(* Logix 5000 project; controller Comas_L4 vendor 1 type 14 code 193 rev 30.11; software revision 30.02; part 11 of 12 *)
(* tags used below, declared in another part *)
   AOI_Badge : Badges_Acces;
   AOI_Cam_Display_Horiz : AOI_CamDisplay_OCX_StdCAM;
   AOI_Cam_Display_Verti : AOI_CamDisplay_OCX_StdCAM;
   AOI_Pilotage_Codeur_Vitesse_Moy : Pilotage_Vitesse_Rapide_V4;
   Axe_Codeur_Four : AXIS_CIP_DRIVE;
   Axe_Horizontal_Gauche : AXIS_CIP_DRIVE;
   Axe_Virtuel_Codeur : AXIS_VIRTUAL;
   Axe_Virtuel_Maitre : AXIS_VIRTUAL;
   Badge_Code_A : BOOL;
   Badge_Code_B : BOOL;
   Badge_Code_C : BOOL;
   Badge_Code_D : BOOL;
   BP_O_F_Trappe : BOOL;
   Cam_Chart_Horiz : Chart;
   Cam_Chart_Verti : Chart;
   Cam_Display_Horiz : UDT_Axis_Cam_Profil;
   Cam_Display_Verti : UDT_Axis_Cam_Profil;
   CO_Acquit_defaut : BOOL;
   CO_Defaut_Four : BOOL;
   CO_Defaut_Relais_Securite : BOOL;
   CO_Defauts_Secondaires : BOOL;
   CO_demande_darret : BOOL;
   CO_en_Marche : BOOL;
   CO_Engage_Axe_H_Droit : Engage_Axe;
   CO_Engage_Axe_H_Gauche : Engage_Axe;
   CO_Engage_Axe_V_Droit : Engage_Axe;
   CO_Engage_Axe_V_Gauche : Engage_Axe;
   CO_Engage_Maitre : Engage_Axe_Virtuel;
   CO_Engagement : BOOL;
   CO_Flip_100ms : TIMER;
   CO_Flip_500ms : TIMER;
   CO_Flop_100ms : TIMER;
   CO_Flop_500ms : TIMER;
   CO_Init_Ok : BOOL;
   CO_Machine_sans_defaut : BOOL;
   CO_Marche : BOOL;
   CO_Pilotage_Coupe_Fil : Pilotage_Relatif_Virtuel;
   CO_Synchro_Axe_En_Cours : BOOL;
   CO_Temps_de_demarrage : TIMER;
   CO_TOF_Top_Decoreuse : TIMER;
   CO_TOF_Top_Doseuse : TIMER;
   CO_Top_Debut_Cycle_Decoreuse : BOOL;
   CO_Top_Debut_Dosage : BOOL;
   CO_Top_Once_Decoreuse : BOOL;
   CO_Top_Once_Doseuse : BOOL;
   CO_Top_Recalage : BOOL;
   Com_Comas_Conv : DINT[10];
   Com_Comas_Gen_Conv : DINT[10];
   Com_Comas_Sortie_F : UDT_COM_Comas_Vers_SortieF;
   Det_Produit : BOOL;
   Det_Produit2 : BOOL;
   ENT_Badge_Code_A : ALIAS FOR Local:1:I.Pt11.Data;
   ENT_Badge_Code_B : ALIAS FOR Local:1:I.Pt12.Data;
   ENT_Badge_Code_C : ALIAS FOR Local:1:I.Pt13.Data;
   ENT_Badge_Code_D : ALIAS FOR Local:1:I.Pt14.Data;
   ENT_Badge_STR : ALIAS FOR Local:1:I.Pt15.Data;
   ENT_CO_BP_Arret : ALIAS FOR Local:1:I.Pt01.Data;
   ENT_CO_BP_Marche : ALIAS FOR Local:1:I.Pt00.Data;
   ENT_Reisdorf_en_Marche : ALIAS FOR Local:2:I.Pt03.Data;
   Fin_Rouleau : REAL;
   Flip_Display : TIMER;
   Flop_Display : TIMER;
   Front_Badge : BOOL;
   Front_Det_produit_Moyennage : BOOL;
   Front_Det_produit_Moyennage2 : BOOL;
   Front_Resynchro_temp : BOOL;
   Front_Top_Recalage : BOOL;
   Lecteur_Badge_Code_A : BOOL;
   Lecteur_Badge_Code_B : BOOL;
   Lecteur_Badge_Code_C : BOOL;
   Lecteur_Badge_Code_D : BOOL;
   MAM_Resyncho_Codeur : MOTION_INSTRUCTION;
   MAM_Resynchro_Accel_Correction : REAL;
   MAM_Resynchro_Vitesse_Correction : REAL;
   Memo_Recalage_Detection_PRoduit_1 : BOOL;
   Memo_Recalage_Detection_PRoduit_2 : BOOL;
   MSG_General_Convoyage : MESSAGE;
   MSG_Vitesse_Four_L4 : MESSAGE;
   Output_Cams_Decoreuse : Output_Cams;
   Output_Cams_Dosage : Output_Cams;
   Output_Cams_Recalage : Output_Cams;
   PCAM_Horizontal : UDT_CamGeneration;
   PCAM_Vertical : UDT_CamGeneration;
   Position_Codeur_Virtuel_Det_Produit : REAL;
   Position_Decalee : REAL;
   RECETTE_EC : UDT_RECIPE;
   Resynchro_Codeur : BOOL;
   Resynchro_Codeur_Front : BOOL;
   RSW_BADGE_Numero_Page : DINT;
   RSW_BADGE_Numero_Page_En_Cours : DINT;
   RSW_BADGE_RAZ_CODE : BOOL;
   RSW_BADGE_Temps_Restant : DINT;
   RSW_BADGE_TOF_Chagement_Page : TIMER;
   RSW_Niveau_Accu_LA : DINT;
   RSW_Niveau_Accu_LD : DINT;
   SOR_CO_Echange_Amont_OK : ALIAS FOR Local:3:O.Pt07.Data;
   SOR_CO_Top_Debut_Cycle_Decoreuse : ALIAS FOR Local:3:O.Pt05.Data;
   SOR_CO_Top_Debut_Dosage : ALIAS FOR Local:3:O.Pt06.Data;
   SOR_CO_Voyant_Arret : ALIAS FOR Local:3:O.Pt01.Data;
   SOR_CO_Voyant_Marche : ALIAS FOR Local:3:O.Pt00.Data;
   SOR_CO_Voyant_Rearmement : ALIAS FOR Local:3:O.Pt02.Data;
   Speed_Control_Pompe : Axis_speed_control;
   Start_Cam_Logique_Rouleaux : REAL;
   Stop_Cam_Logique_Rouleaux : REAL;
   Tab_Position_Correction : REAL[50];
   Tab_Position_Correction_Temp : REAL[50];
   Temps_total_avant_arret_L4 : REAL;
   TimeOutResynch_Codeur : TIMER;
   TON_Simul_Produit : TIMER;
   Val_Position_Recalage : REAL;
   Val_Position_Recalage_Tab1 : REAL;
   Val_Position_Recalage_Tab2 : REAL;
   Val_Position_Recalage_Tab3 : REAL;
   Val_Position_Recalage_Tab4 : REAL;
   Val_Position_Recalage_Tab5 : REAL;
   Vitesse_Four4_Real : REAL;
(* General, continued *)

ROUTINE D00_Marche   (* ladder *)
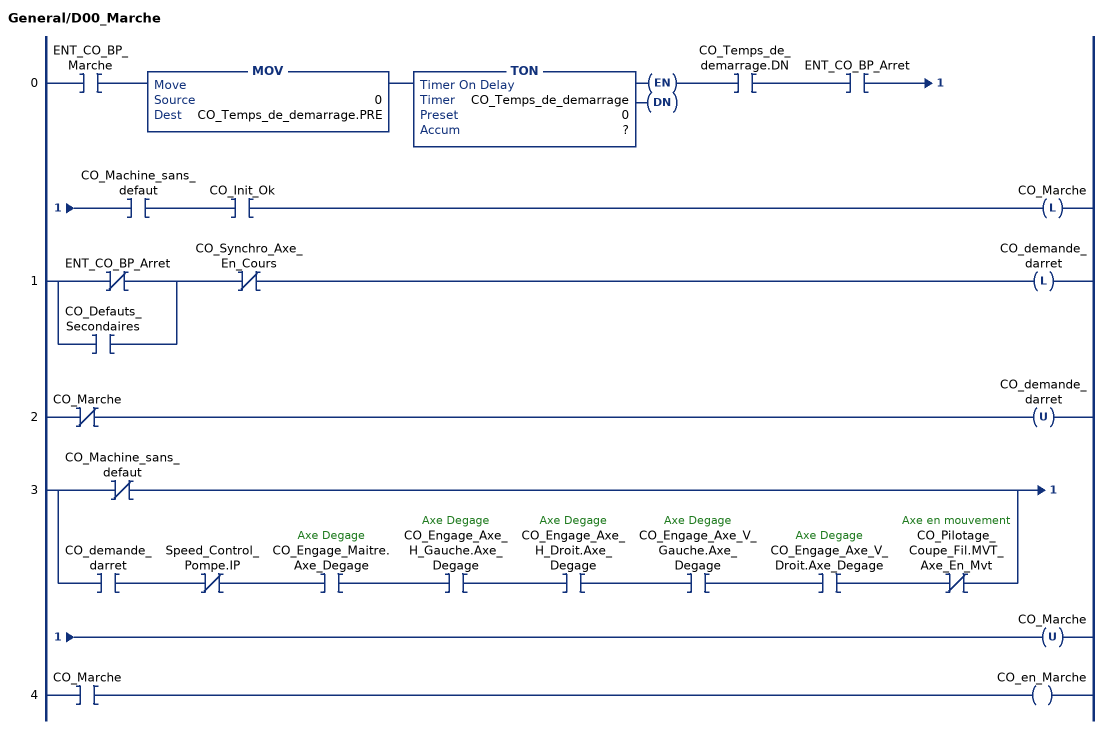
   0: XIC(ENT_CO_BP_Marche)MOV(0,CO_Temps_de_demarrage.PRE)TON(CO_Temps_de_demarrage,?,?)XIC(CO_Temps_de_demarrage.DN)XIC(ENT_CO_BP_Arret)XIC(CO_Machine_sans_defaut)XIC(CO_Init_Ok)OTL(CO_Marche);
   1: [XIO(ENT_CO_BP_Arret) ,XIC(CO_Defauts_Secondaires) ]XIO(CO_Synchro_Axe_En_Cours)OTL(CO_demande_darret);
   2: XIO(CO_Marche)OTU(CO_demande_darret);
   3: [XIO(CO_Machine_sans_defaut) ,XIC(CO_demande_darret) XIO(Speed_Control_Pompe.IP) XIC(CO_Engage_Maitre.Axe_Degage) XIC(CO_Engage_Axe_H_Gauche.Axe_Degage) XIC(CO_Engage_Axe_H_Droit.Axe_Degage) XIC(CO_Engage_Axe_V_Gauche.Axe_Degage) XIC(CO_Engage_Axe_V_Droit.Axe_Degage) XIO(CO_Pilotage_Coupe_Fil.MVT_Axe_En_Mvt) ]OTU(CO_Marche);
   4: XIC(CO_Marche)OTE(CO_en_Marche);
END_ROUTINE

ROUTINE E00_Voyants   (* ladder *)
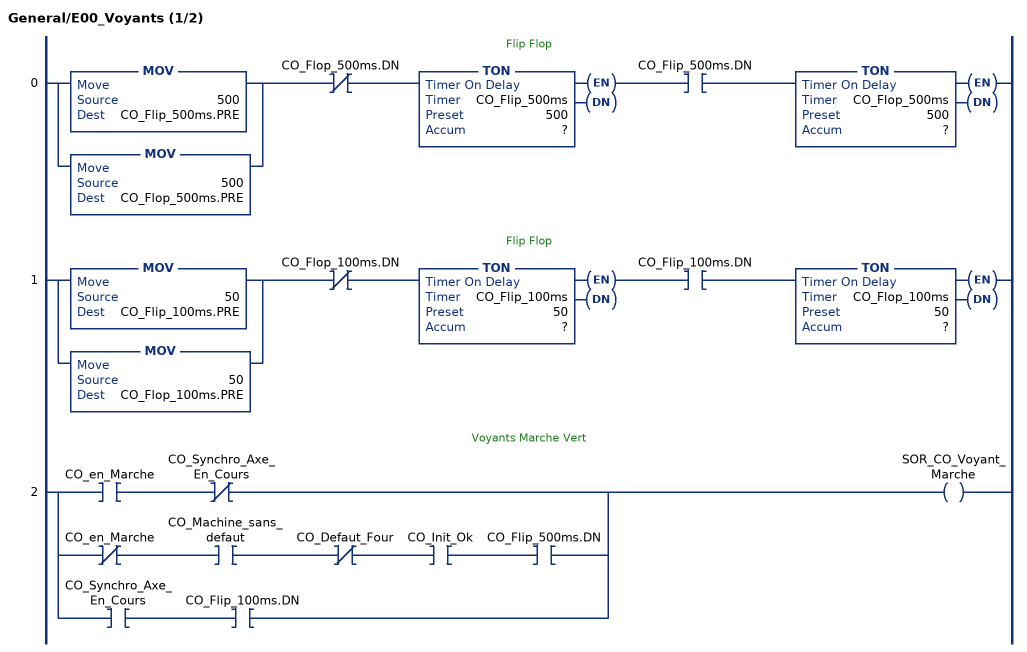
   // Flip Flop
   0: [MOV(500,CO_Flip_500ms.PRE) ,MOV(500,CO_Flop_500ms.PRE) ]XIO(CO_Flop_500ms.DN)TON(CO_Flip_500ms,?,?)XIC(CO_Flip_500ms.DN)TON(CO_Flop_500ms,?,?);
   // Flip Flop
   1: [MOV(50,CO_Flip_100ms.PRE) ,MOV(50,CO_Flop_100ms.PRE) ]XIO(CO_Flop_100ms.DN)TON(CO_Flip_100ms,?,?)XIC(CO_Flip_100ms.DN)TON(CO_Flop_100ms,?,?);
   // Voyants Marche Vert
   2: [XIC(CO_en_Marche) XIO(CO_Synchro_Axe_En_Cours) ,XIO(CO_en_Marche) XIC(CO_Machine_sans_defaut) XIO(CO_Defaut_Four) XIC(CO_Init_Ok) XIC(CO_Flip_500ms.DN) ,XIC(CO_Synchro_Axe_En_Cours) XIC(CO_Flip_100ms.DN) ]OTE(SOR_CO_Voyant_Marche);
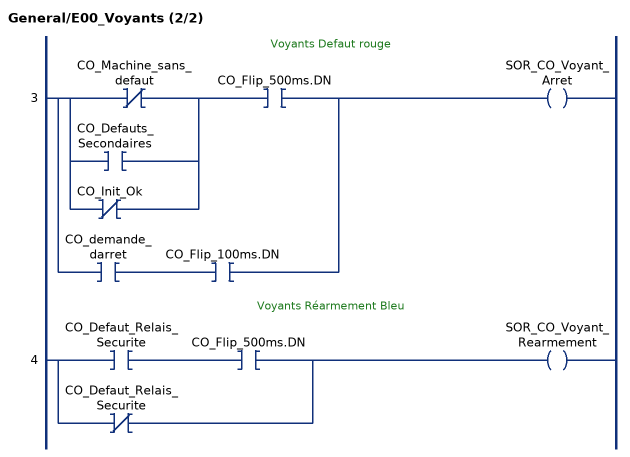
   // Voyants Defaut rouge
   3: [[XIO(CO_Machine_sans_defaut) ,XIC(CO_Defauts_Secondaires) ,XIO(CO_Init_Ok) ] XIC(CO_Flip_500ms.DN) ,XIC(CO_demande_darret) XIC(CO_Flip_100ms.DN) ]OTE(SOR_CO_Voyant_Arret);
   // Voyants Réarmement Bleu
   4: [XIC(CO_Defaut_Relais_Securite) XIC(CO_Flip_500ms.DN) ,XIO(CO_Defaut_Relais_Securite) ]OTE(SOR_CO_Voyant_Rearmement);
END_ROUTINE

ROUTINE Z00_EXT   (* ladder *)
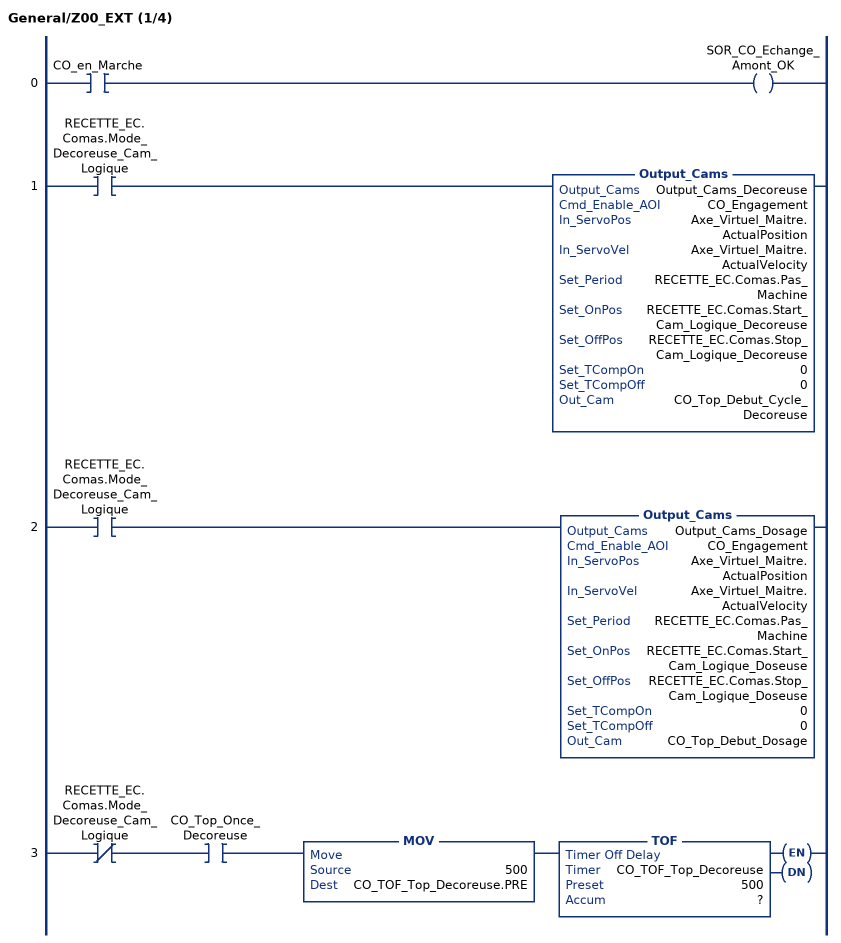
   0: XIC(CO_en_Marche)OTE(SOR_CO_Echange_Amont_OK);
   1: XIC(RECETTE_EC.Comas.Mode_Decoreuse_Cam_Logique)Output_Cams(Output_Cams_Decoreuse,CO_Engagement,Axe_Virtuel_Maitre.ActualPosition,Axe_Virtuel_Maitre.ActualVelocity,RECETTE_EC.Comas.Pas_Machine,RECETTE_EC.Comas.Start_Cam_Logique_Decoreuse,RECETTE_EC.Comas.Stop_Cam_Logique_Decoreuse,0,0,CO_Top_Debut_Cycle_Decoreuse);
   2: XIC(RECETTE_EC.Comas.Mode_Decoreuse_Cam_Logique)Output_Cams(Output_Cams_Dosage,CO_Engagement,Axe_Virtuel_Maitre.ActualPosition,Axe_Virtuel_Maitre.ActualVelocity,RECETTE_EC.Comas.Pas_Machine,RECETTE_EC.Comas.Start_Cam_Logique_Doseuse,RECETTE_EC.Comas.Stop_Cam_Logique_Doseuse,0,0,CO_Top_Debut_Dosage);
   3: XIO(RECETTE_EC.Comas.Mode_Decoreuse_Cam_Logique)XIC(CO_Top_Once_Decoreuse)MOV(500,CO_TOF_Top_Decoreuse.PRE)TOF(CO_TOF_Top_Decoreuse,?,?);
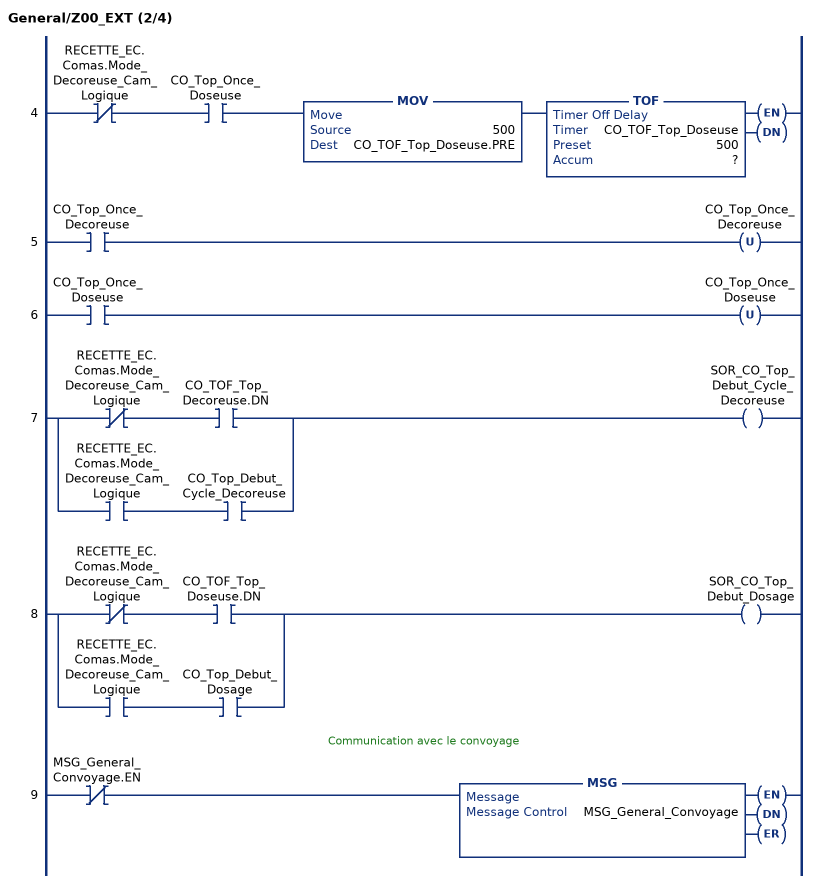
   4: XIO(RECETTE_EC.Comas.Mode_Decoreuse_Cam_Logique)XIC(CO_Top_Once_Doseuse)MOV(500,CO_TOF_Top_Doseuse.PRE)TOF(CO_TOF_Top_Doseuse,?,?);
   5: XIC(CO_Top_Once_Decoreuse)OTU(CO_Top_Once_Decoreuse);
   6: XIC(CO_Top_Once_Doseuse)OTU(CO_Top_Once_Doseuse);
   7: [XIO(RECETTE_EC.Comas.Mode_Decoreuse_Cam_Logique) XIC(CO_TOF_Top_Decoreuse.DN) ,XIC(RECETTE_EC.Comas.Mode_Decoreuse_Cam_Logique) XIC(CO_Top_Debut_Cycle_Decoreuse) ]OTE(SOR_CO_Top_Debut_Cycle_Decoreuse);
   8: [XIO(RECETTE_EC.Comas.Mode_Decoreuse_Cam_Logique) XIC(CO_TOF_Top_Doseuse.DN) ,XIC(RECETTE_EC.Comas.Mode_Decoreuse_Cam_Logique) XIC(CO_Top_Debut_Dosage) ]OTE(SOR_CO_Top_Debut_Dosage);
   // Communication avec le convoyage
   9: XIO(MSG_General_Convoyage.EN)MSG(MSG_General_Convoyage);
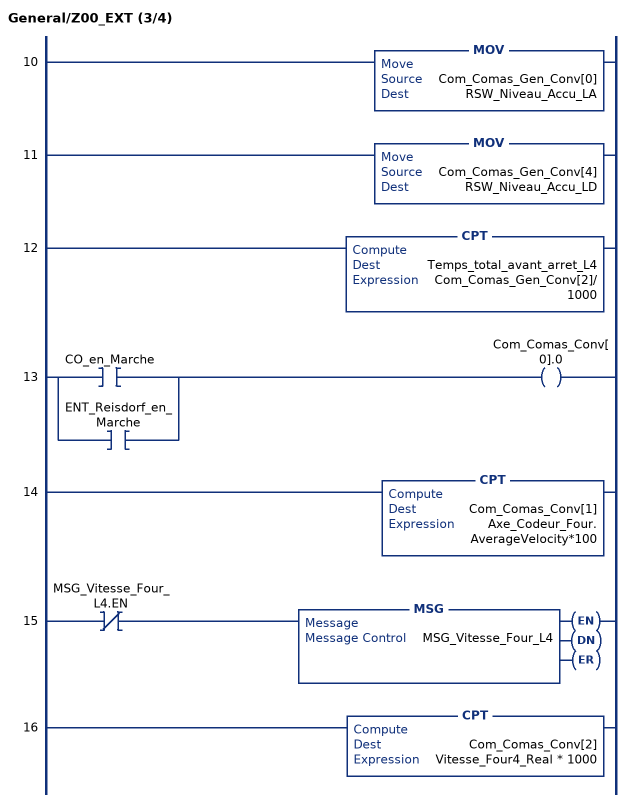
   10: MOV(Com_Comas_Gen_Conv[0],RSW_Niveau_Accu_LA);
   11: MOV(Com_Comas_Gen_Conv[4],RSW_Niveau_Accu_LD);
   12: CPT(Temps_total_avant_arret_L4,Com_Comas_Gen_Conv[2]/1000);
   13: [XIC(CO_en_Marche) ,XIC(ENT_Reisdorf_en_Marche) ]OTE(Com_Comas_Conv[0].0);
   14: CPT(Com_Comas_Conv[1],Axe_Codeur_Four.AverageVelocity*100);
   15: XIO(MSG_Vitesse_Four_L4.EN)MSG(MSG_Vitesse_Four_L4);
   16: CPT(Com_Comas_Conv[2],Vitesse_Four4_Real * 1000);
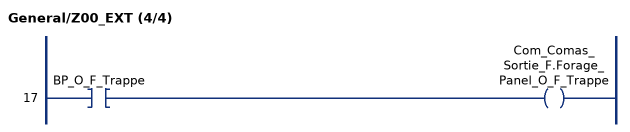
   17: XIC(BP_O_F_Trappe)OTE(Com_Comas_Sortie_F.Forage_Panel_O_F_Trappe);
END_ROUTINE

ROUTINE Z01_Badges_Acc   (* ladder *)
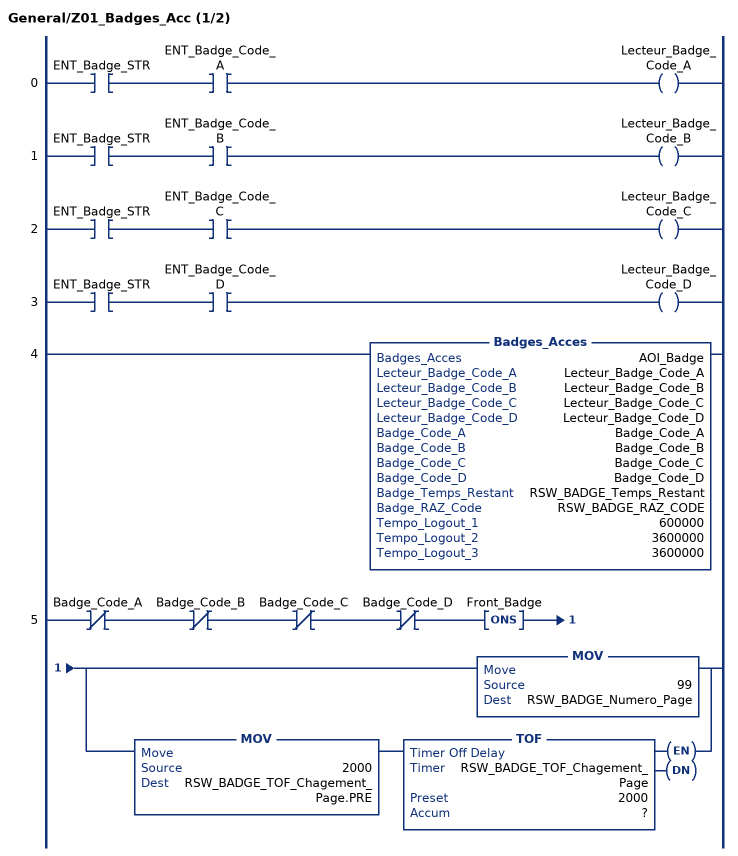
   0: XIC(ENT_Badge_STR)XIC(ENT_Badge_Code_A)OTE(Lecteur_Badge_Code_A);
   1: XIC(ENT_Badge_STR)XIC(ENT_Badge_Code_B)OTE(Lecteur_Badge_Code_B);
   2: XIC(ENT_Badge_STR)XIC(ENT_Badge_Code_C)OTE(Lecteur_Badge_Code_C);
   3: XIC(ENT_Badge_STR)XIC(ENT_Badge_Code_D)OTE(Lecteur_Badge_Code_D);
   4: Badges_Acces(AOI_Badge,Lecteur_Badge_Code_A,Lecteur_Badge_Code_B,Lecteur_Badge_Code_C,Lecteur_Badge_Code_D,Badge_Code_A,Badge_Code_B,Badge_Code_C,Badge_Code_D,RSW_BADGE_Temps_Restant,RSW_BADGE_RAZ_CODE,600000,3600000,3600000);
   5: XIO(Badge_Code_A)XIO(Badge_Code_B)XIO(Badge_Code_C)XIO(Badge_Code_D)ONS(Front_Badge)[MOV(99,RSW_BADGE_Numero_Page) ,MOV(2000,RSW_BADGE_TOF_Chagement_Page.PRE) TOF(RSW_BADGE_TOF_Chagement_Page,?,?) ];
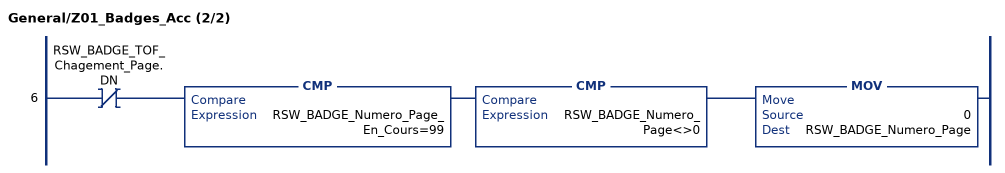
   6: XIO(RSW_BADGE_TOF_Chagement_Page.DN)CMP(RSW_BADGE_Numero_Page_En_Cours=99)CMP(RSW_BADGE_Numero_Page<>0)MOV(0,RSW_BADGE_Numero_Page);
END_ROUTINE

ROUTINE Z02_Cames   (* ladder *)
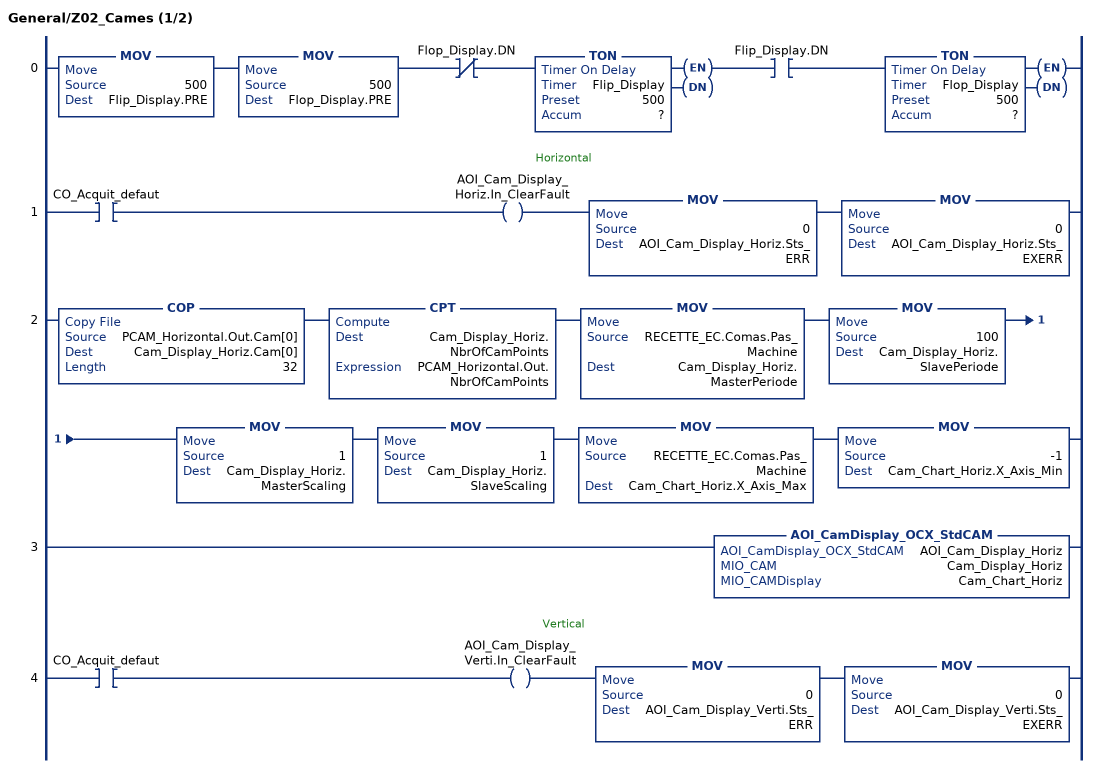
   0: MOV(500,Flip_Display.PRE)MOV(500,Flop_Display.PRE)XIO(Flop_Display.DN)TON(Flip_Display,?,?)XIC(Flip_Display.DN)TON(Flop_Display,?,?);
   // Horizontal
   1: XIC(CO_Acquit_defaut)OTE(AOI_Cam_Display_Horiz.In_ClearFault)MOV(0,AOI_Cam_Display_Horiz.Sts_ERR)MOV(0,AOI_Cam_Display_Horiz.Sts_EXERR);
   2: COP(PCAM_Horizontal.Out.Cam[0],Cam_Display_Horiz.Cam[0],32)CPT(Cam_Display_Horiz.NbrOfCamPoints,PCAM_Horizontal.Out.NbrOfCamPoints)MOV(RECETTE_EC.Comas.Pas_Machine,Cam_Display_Horiz.MasterPeriode)MOV(100,Cam_Display_Horiz.SlavePeriode)MOV(1,Cam_Display_Horiz.MasterScaling)MOV(1,Cam_Display_Horiz.SlaveScaling)MOV(RECETTE_EC.Comas.Pas_Machine,Cam_Chart_Horiz.X_Axis_Max)MOV(-1,Cam_Chart_Horiz.X_Axis_Min);
   3: AOI_CamDisplay_OCX_StdCAM(AOI_Cam_Display_Horiz,Cam_Display_Horiz,Cam_Chart_Horiz);
   // Vertical
   4: XIC(CO_Acquit_defaut)OTE(AOI_Cam_Display_Verti.In_ClearFault)MOV(0,AOI_Cam_Display_Verti.Sts_ERR)MOV(0,AOI_Cam_Display_Verti.Sts_EXERR);
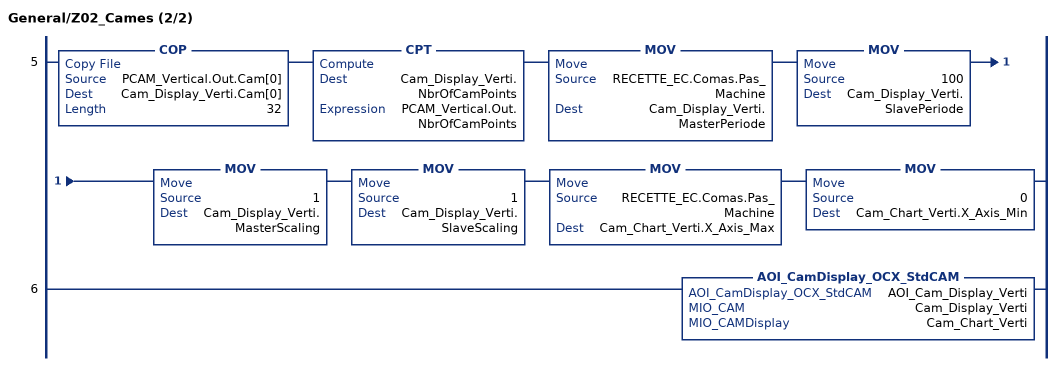
   5: COP(PCAM_Vertical.Out.Cam[0],Cam_Display_Verti.Cam[0],32)CPT(Cam_Display_Verti.NbrOfCamPoints,PCAM_Vertical.Out.NbrOfCamPoints)MOV(RECETTE_EC.Comas.Pas_Machine,Cam_Display_Verti.MasterPeriode)MOV(100,Cam_Display_Verti.SlavePeriode)MOV(1,Cam_Display_Verti.MasterScaling)MOV(1,Cam_Display_Verti.SlaveScaling)MOV(RECETTE_EC.Comas.Pas_Machine,Cam_Chart_Verti.X_Axis_Max)MOV(0,Cam_Chart_Verti.X_Axis_Min);
   6: AOI_CamDisplay_OCX_StdCAM(AOI_Cam_Display_Verti,Cam_Display_Verti,Cam_Chart_Verti);
END_ROUTINE
END_PROGRAM

PROGRAM Main   (* main routine A00_Appel *)

ROUTINE A00_Appel   (* ladder *)
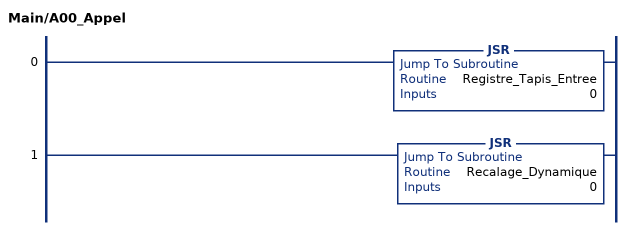
   0: JSR(Registre_Tapis_Entree,0);
   1: JSR(Recalage_Dynamique,0);
END_ROUTINE

ROUTINE Recalage_Dynamique   (* ladder *)
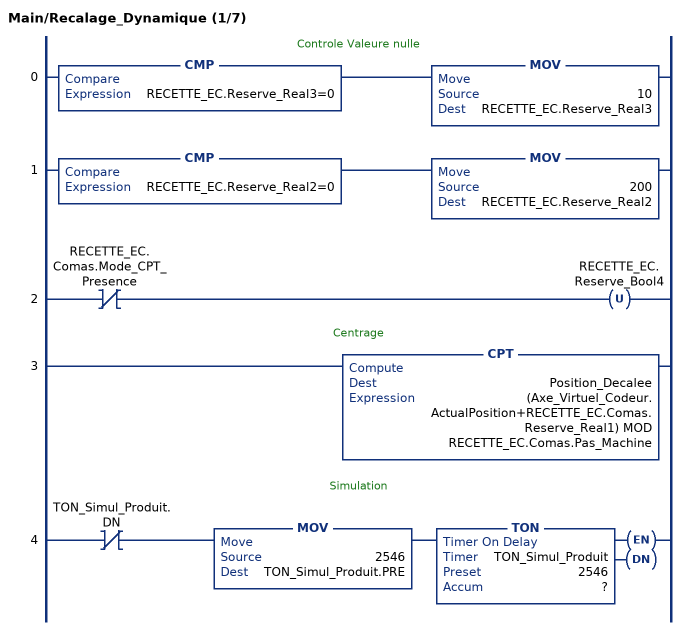
   // Controle Valeure nulle
   0: CMP(RECETTE_EC.Reserve_Real3=0)MOV(10,RECETTE_EC.Reserve_Real3);
   1: CMP(RECETTE_EC.Reserve_Real2=0)MOV(200,RECETTE_EC.Reserve_Real2);
   2: XIO(RECETTE_EC.Comas.Mode_CPT_Presence)OTU(RECETTE_EC.Reserve_Bool4);
   // Centrage
   3: CPT(Position_Decalee,(Axe_Virtuel_Codeur.ActualPosition+RECETTE_EC.Comas.Reserve_Real1) MOD RECETTE_EC.Comas.Pas_Machine);
   // Simulation
   4: XIO(TON_Simul_Produit.DN)MOV(2546,TON_Simul_Produit.PRE)TON(TON_Simul_Produit,?,?);
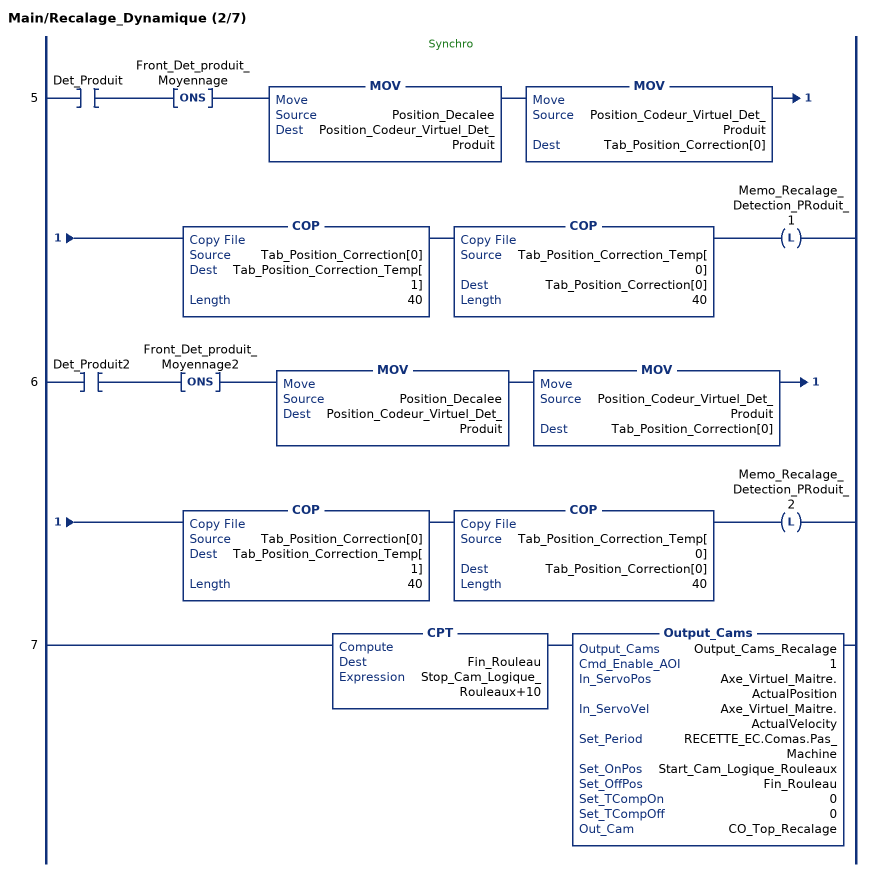
   // Synchro
   5: XIC(Det_Produit)ONS(Front_Det_produit_Moyennage)MOV(Position_Decalee,Position_Codeur_Virtuel_Det_Produit)MOV(Position_Codeur_Virtuel_Det_Produit,Tab_Position_Correction[0])COP(Tab_Position_Correction[0],Tab_Position_Correction_Temp[1],40)COP(Tab_Position_Correction_Temp[0],Tab_Position_Correction[0],40)OTL(Memo_Recalage_Detection_PRoduit_1);
   6: XIC(Det_Produit2)ONS(Front_Det_produit_Moyennage2)MOV(Position_Decalee,Position_Codeur_Virtuel_Det_Produit)MOV(Position_Codeur_Virtuel_Det_Produit,Tab_Position_Correction[0])COP(Tab_Position_Correction[0],Tab_Position_Correction_Temp[1],40)COP(Tab_Position_Correction_Temp[0],Tab_Position_Correction[0],40)OTL(Memo_Recalage_Detection_PRoduit_2);
   7: CPT(Fin_Rouleau,Stop_Cam_Logique_Rouleaux+10)Output_Cams(Output_Cams_Recalage,1,Axe_Virtuel_Maitre.ActualPosition,Axe_Virtuel_Maitre.ActualVelocity,RECETTE_EC.Comas.Pas_Machine,Start_Cam_Logique_Rouleaux,Fin_Rouleau,0,0,CO_Top_Recalage);
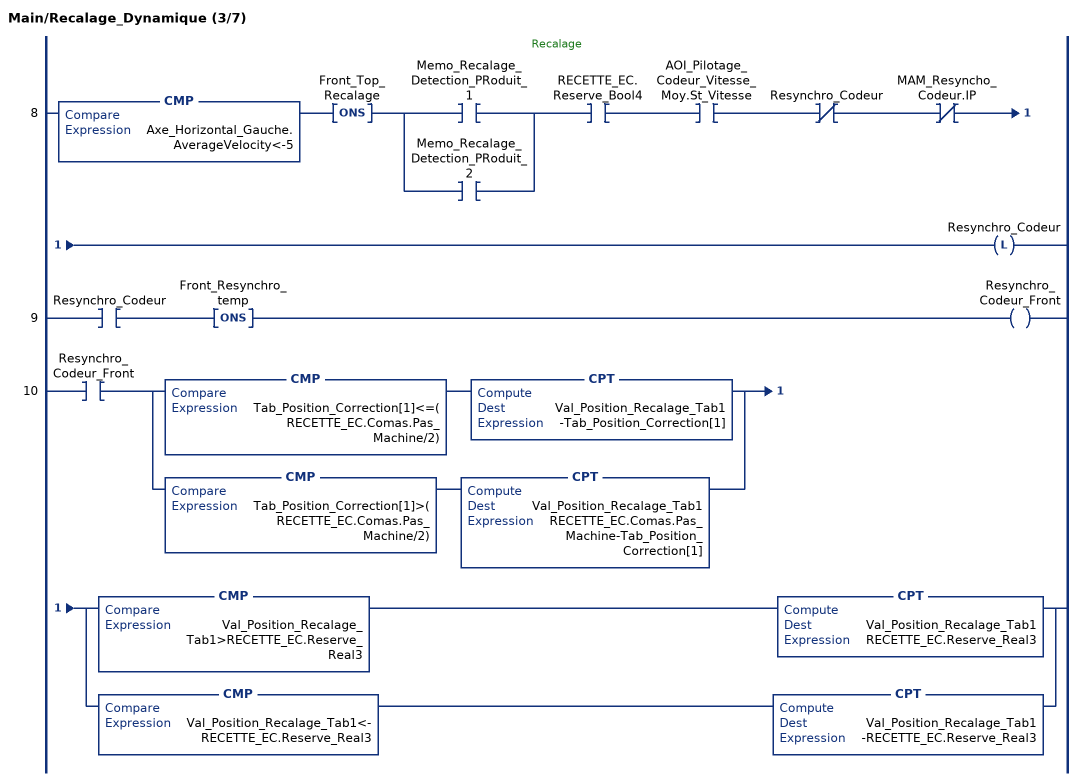
   // Recalage
   8: CMP(Axe_Horizontal_Gauche.AverageVelocity<-5)ONS(Front_Top_Recalage)[XIC(Memo_Recalage_Detection_PRoduit_1) ,XIC(Memo_Recalage_Detection_PRoduit_2) ]XIC(RECETTE_EC.Reserve_Bool4)XIC(AOI_Pilotage_Codeur_Vitesse_Moy.St_Vitesse)XIO(Resynchro_Codeur)XIO(MAM_Resyncho_Codeur.IP)OTL(Resynchro_Codeur);
   9: XIC(Resynchro_Codeur)ONS(Front_Resynchro_temp)OTE(Resynchro_Codeur_Front);
   10: XIC(Resynchro_Codeur_Front)[CMP(Tab_Position_Correction[1]<=(RECETTE_EC.Comas.Pas_Machine/2)) CPT(Val_Position_Recalage_Tab1,-Tab_Position_Correction[1]) ,CMP(Tab_Position_Correction[1]>(RECETTE_EC.Comas.Pas_Machine/2)) CPT(Val_Position_Recalage_Tab1,RECETTE_EC.Comas.Pas_Machine-Tab_Position_Correction[1]) ][CMP(Val_Position_Recalage_Tab1>RECETTE_EC.Reserve_Real3) CPT(Val_Position_Recalage_Tab1,RECETTE_EC.Reserve_Real3) ,CMP(Val_Position_Recalage_Tab1<-RECETTE_EC.Reserve_Real3) CPT(Val_Position_Recalage_Tab1,-RECETTE_EC.Reserve_Real3) ];
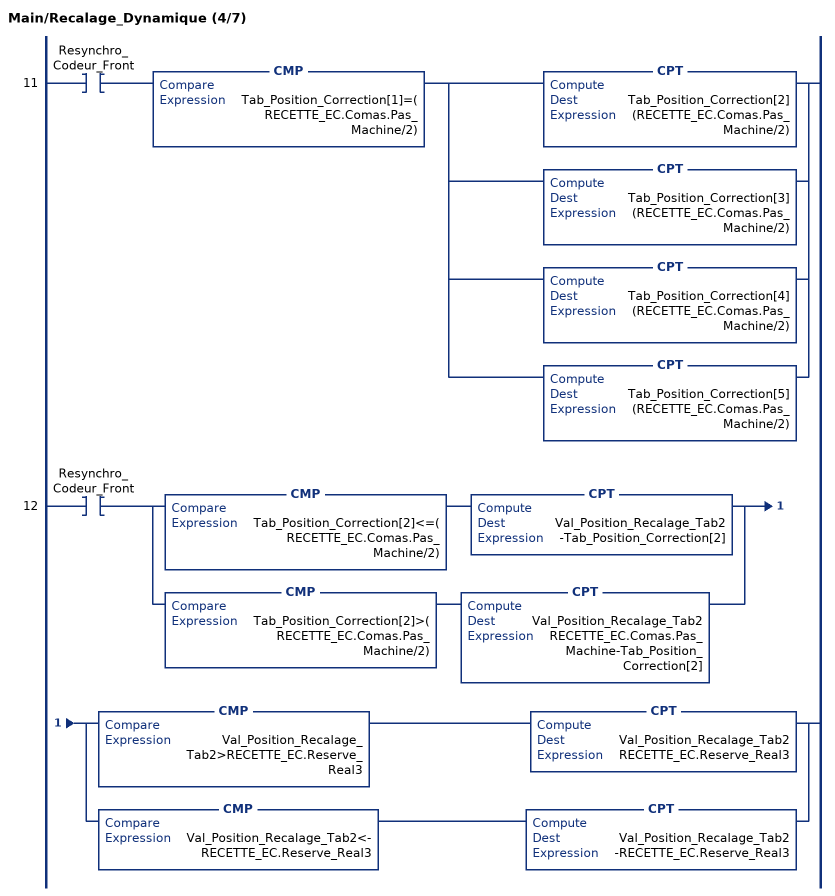
   11: XIC(Resynchro_Codeur_Front)CMP(Tab_Position_Correction[1]=(RECETTE_EC.Comas.Pas_Machine/2))[CPT(Tab_Position_Correction[2],(RECETTE_EC.Comas.Pas_Machine/2)) ,CPT(Tab_Position_Correction[3],(RECETTE_EC.Comas.Pas_Machine/2)) ,CPT(Tab_Position_Correction[4],(RECETTE_EC.Comas.Pas_Machine/2)) ,CPT(Tab_Position_Correction[5],(RECETTE_EC.Comas.Pas_Machine/2)) ];
   12: XIC(Resynchro_Codeur_Front)[CMP(Tab_Position_Correction[2]<=(RECETTE_EC.Comas.Pas_Machine/2)) CPT(Val_Position_Recalage_Tab2,-Tab_Position_Correction[2]) ,CMP(Tab_Position_Correction[2]>(RECETTE_EC.Comas.Pas_Machine/2)) CPT(Val_Position_Recalage_Tab2,RECETTE_EC.Comas.Pas_Machine-Tab_Position_Correction[2]) ][CMP(Val_Position_Recalage_Tab2>RECETTE_EC.Reserve_Real3) CPT(Val_Position_Recalage_Tab2,RECETTE_EC.Reserve_Real3) ,CMP(Val_Position_Recalage_Tab2<-RECETTE_EC.Reserve_Real3) CPT(Val_Position_Recalage_Tab2,-RECETTE_EC.Reserve_Real3) ];
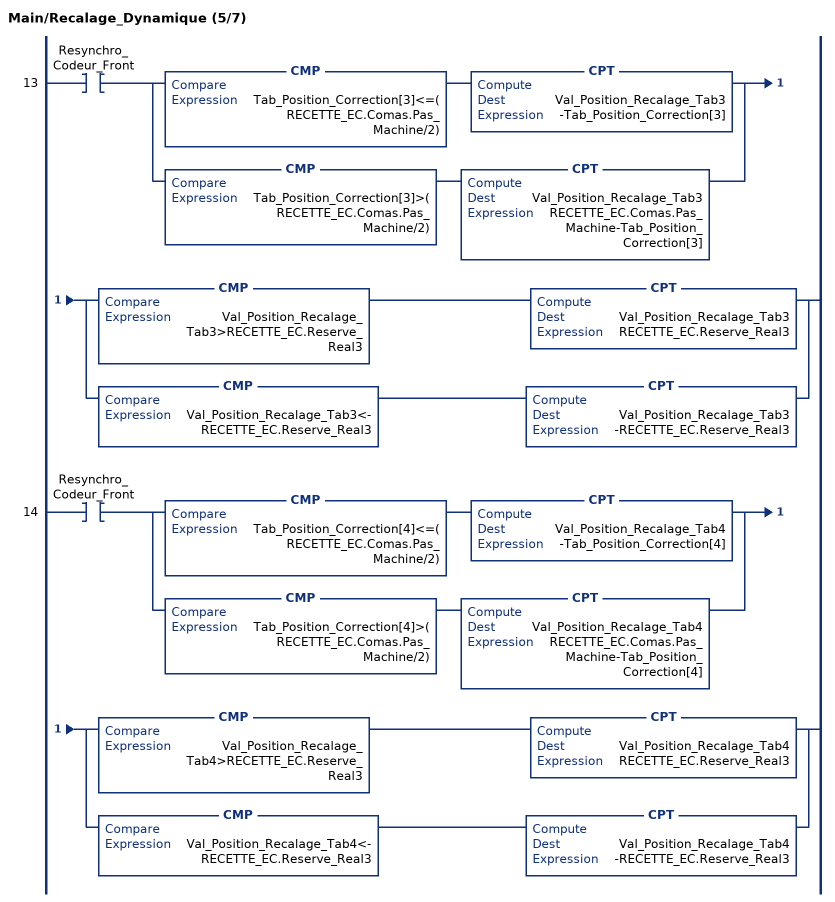
   13: XIC(Resynchro_Codeur_Front)[CMP(Tab_Position_Correction[3]<=(RECETTE_EC.Comas.Pas_Machine/2)) CPT(Val_Position_Recalage_Tab3,-Tab_Position_Correction[3]) ,CMP(Tab_Position_Correction[3]>(RECETTE_EC.Comas.Pas_Machine/2)) CPT(Val_Position_Recalage_Tab3,RECETTE_EC.Comas.Pas_Machine-Tab_Position_Correction[3]) ][CMP(Val_Position_Recalage_Tab3>RECETTE_EC.Reserve_Real3) CPT(Val_Position_Recalage_Tab3,RECETTE_EC.Reserve_Real3) ,CMP(Val_Position_Recalage_Tab3<-RECETTE_EC.Reserve_Real3) CPT(Val_Position_Recalage_Tab3,-RECETTE_EC.Reserve_Real3) ];
   14: XIC(Resynchro_Codeur_Front)[CMP(Tab_Position_Correction[4]<=(RECETTE_EC.Comas.Pas_Machine/2)) CPT(Val_Position_Recalage_Tab4,-Tab_Position_Correction[4]) ,CMP(Tab_Position_Correction[4]>(RECETTE_EC.Comas.Pas_Machine/2)) CPT(Val_Position_Recalage_Tab4,RECETTE_EC.Comas.Pas_Machine-Tab_Position_Correction[4]) ][CMP(Val_Position_Recalage_Tab4>RECETTE_EC.Reserve_Real3) CPT(Val_Position_Recalage_Tab4,RECETTE_EC.Reserve_Real3) ,CMP(Val_Position_Recalage_Tab4<-RECETTE_EC.Reserve_Real3) CPT(Val_Position_Recalage_Tab4,-RECETTE_EC.Reserve_Real3) ];
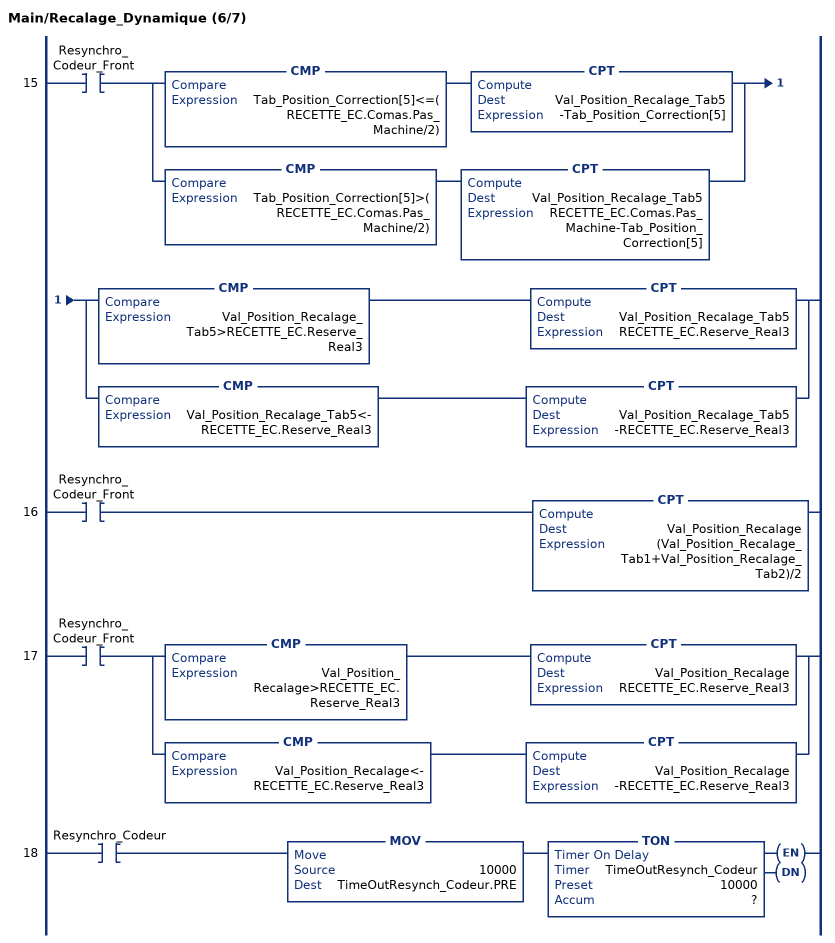
   15: XIC(Resynchro_Codeur_Front)[CMP(Tab_Position_Correction[5]<=(RECETTE_EC.Comas.Pas_Machine/2)) CPT(Val_Position_Recalage_Tab5,-Tab_Position_Correction[5]) ,CMP(Tab_Position_Correction[5]>(RECETTE_EC.Comas.Pas_Machine/2)) CPT(Val_Position_Recalage_Tab5,RECETTE_EC.Comas.Pas_Machine-Tab_Position_Correction[5]) ][CMP(Val_Position_Recalage_Tab5>RECETTE_EC.Reserve_Real3) CPT(Val_Position_Recalage_Tab5,RECETTE_EC.Reserve_Real3) ,CMP(Val_Position_Recalage_Tab5<-RECETTE_EC.Reserve_Real3) CPT(Val_Position_Recalage_Tab5,-RECETTE_EC.Reserve_Real3) ];
   16: XIC(Resynchro_Codeur_Front)CPT(Val_Position_Recalage,(Val_Position_Recalage_Tab1+Val_Position_Recalage_Tab2)/2);
   17: XIC(Resynchro_Codeur_Front)[CMP(Val_Position_Recalage>RECETTE_EC.Reserve_Real3) CPT(Val_Position_Recalage,RECETTE_EC.Reserve_Real3) ,CMP(Val_Position_Recalage<-RECETTE_EC.Reserve_Real3) CPT(Val_Position_Recalage,-RECETTE_EC.Reserve_Real3) ];
   18: XIC(Resynchro_Codeur)MOV(10000,TimeOutResynch_Codeur.PRE)TON(TimeOutResynch_Codeur,?,?);
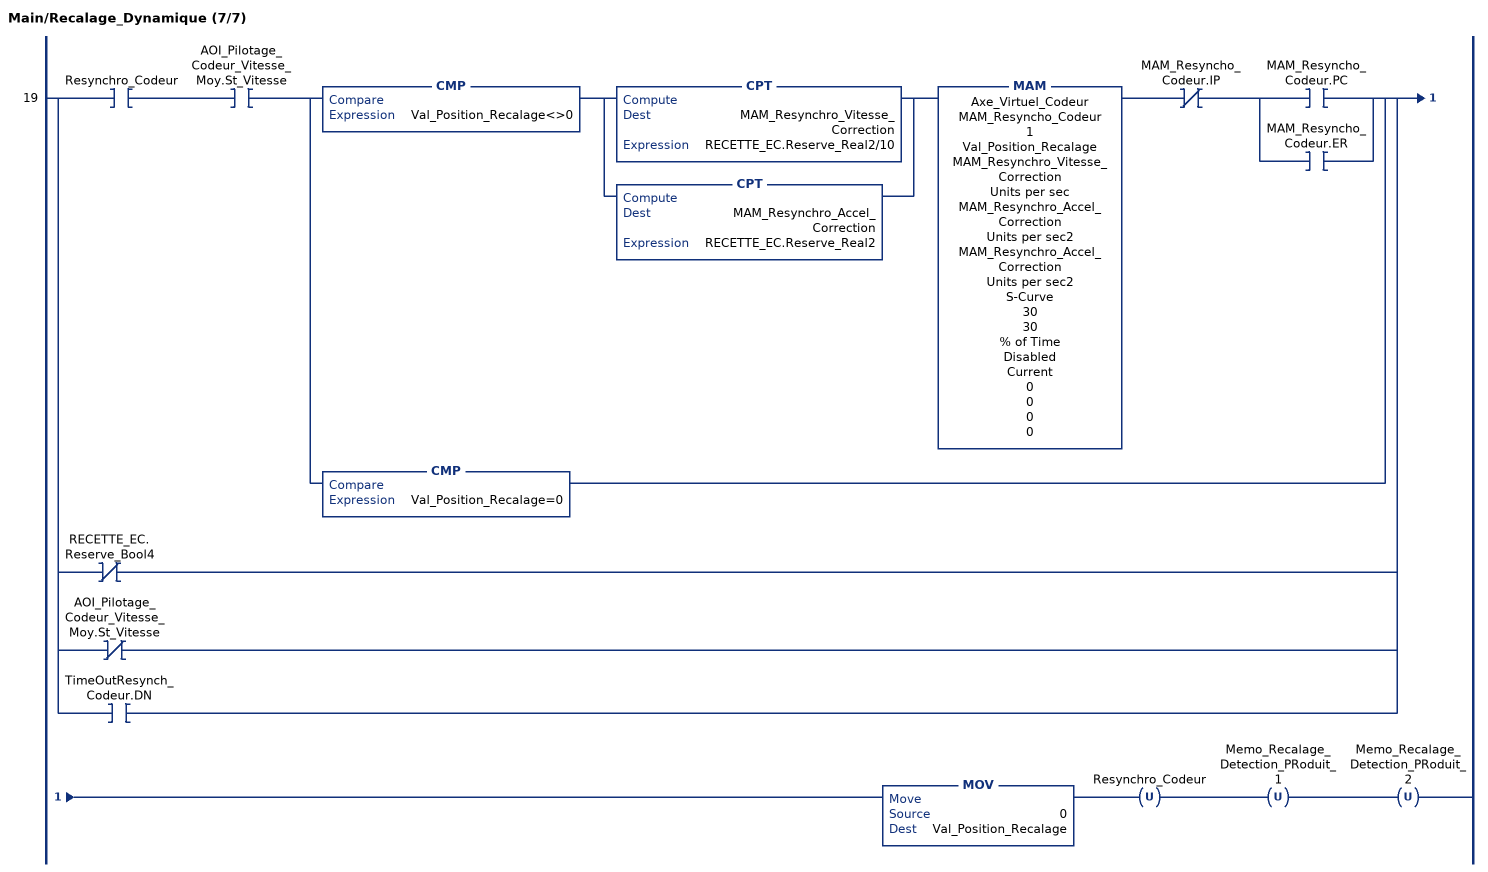
   19: [XIC(Resynchro_Codeur) XIC(AOI_Pilotage_Codeur_Vitesse_Moy.St_Vitesse) [CMP(Val_Position_Recalage<>0) [CPT(MAM_Resynchro_Vitesse_Correction,RECETTE_EC.Reserve_Real2/10) ,CPT(MAM_Resynchro_Accel_Correction,RECETTE_EC.Reserve_Real2) ] MAM(Axe_Virtuel_Codeur,MAM_Resyncho_Codeur,1,Val_Position_Recalage,MAM_Resynchro_Vitesse_Correction,Units per sec,MAM_Resynchro_Accel_Correction,Units per sec2,MAM_Resynchro_Accel_Correction,Units per sec2,S-Curve,30,30,% of Time,Disabled,Current,0,0,0,0) XIO(MAM_Resyncho_Codeur.IP) [XIC(MAM_Resyncho_Codeur.PC) ,XIC(MAM_Resyncho_Codeur.ER) ] ,CMP(Val_Position_Recalage=0) ] ,[XIO(RECETTE_EC.Reserve_Bool4) ,XIO(AOI_Pilotage_Codeur_Vitesse_Moy.St_Vitesse) ,XIC(TimeOutResynch_Codeur.DN) ] ]MOV(0,Val_Position_Recalage)OTU(Resynchro_Codeur)OTU(Memo_Recalage_Detection_PRoduit_1)OTU(Memo_Recalage_Detection_PRoduit_2);
END_ROUTINE
